Staubli VAL3: _stopCycle.pgx

program _stopCycle()
  local string l_sEmpty
  local num nCycleDone
  local num nCycleToDo
  local string sProgName
begin
  // reset the bit
  // Stop the robot
  stopMove()
  if saveData:bStopToPowerOff
    disablePower()
  endIf
  logMsg("[KERNEL] SUPERVISOR:Cycle>Stop cycle")
  // kill the Task...
  taskKill("Cycle")
  taskKill("Action")
  watch(taskStatus("Cycle")==-1 and taskStatus("Action")==-1,1)
  //
  resetMotion()
  call OnEvent:OnCycleEvent(5)
  // delete the last program
  call processList:getCycle(sProgName,nCycleToDo,nCycleDone,0,1)
  if (nCycleToDo-nCycleDone)<=1
    call processList:loopMode()
  else
    call processList:setCycle(sProgName,nCycleToDo,nCycleDone+1,0,1)
  endIf
end
